PROGRAM MAIN
VAR
END_VAR

END_PROGRAM

(* stored: Version 1.1.0.1
   POU MAIN: Id {0d2fa359-362e-46bd-9d15-d56eea26af41} *)
